// TwinCAT 3 PLC project PLC
// ProgramVersion: 3.1.4026.17
// libraries:
//   Tc2_EtherCAT, * (Beckhoff Automation GmbH)
//   Tc2_Standard, * (Beckhoff Automation GmbH)
//   Tc2_System, * (Beckhoff Automation GmbH)
//   Tc3_Module, * (Beckhoff Automation GmbH)
//   VisuDialogs, * (System)
// project tree:
//   DUTs/00_MainBlocks/ E_SystemStartupSequence.TcDUT
//   DUTs/30_EtherCatDiagnostic/ E_EcDiacStatus.TcDUT (not stored), E_EcGetSlaveName.TcDUT (not stored), E_EcSystemStatus.TcDUT (not stored), ST_EcTerminalDiagInfo.TcDUT (not stored)
//   / GlobalTextList.TcGTLO, ImagePool.TcIPO (not stored), PlcTask.TcTTO, Visualization Manager.TcVMO (not stored), VISU_TASK.TcTTO
//   GVLs/ GVL00_IO.TcGVL, GVL10_VAR_PRG.TcGVL, GVL30_DiagnosticEtherCAT.TcGVL
//   POUs/00_MainBlocks/ MAIN.TcPOU
//   POUs/10_GeneralPlcBlocks/ Blinker.TcPOU, ClockGenerator.TcPOU
//   POUs/10_GeneralPlcBlocks/Components/ FB_Blinker.TcPOU, F_ScaleToByteBeam.TcPOU, F_Scaling.TcPOU
//   POUs/11_TemperatureControl/ TemperatureControl.TcPOU
//   POUs/30_EtherCatDiagnose/Components/ FB_DiagnosticEtherCAT.TcPOU (not stored)
//   POUs/30_EtherCatDiagnose/ DiagnosticEtherCAT.TcPOU (not stored)
//   VISUs/ HmiEtherCatDiagnostic.TcVIS, HmiStartPage.TcVIS
// real-time tasks:
//   TASK PlcTask: cycle T#10ms, priority 20, ADS port 350
//   TASK VISU_TASK: cycle T#200000us, priority 30, ADS port 351
// motion (NC):
//   TASK NC-Task 1 SAF: cycle T#2ms, priority 4, ADS port 501
//   TASK NC-Task 1 SVB: cycle T#10ms, priority 8, ADS port 511
//   AXIS Axis 1 (id 1)
//     OtherSettings: AllowMotionCmdToSlave=true
//     encoder EncType=4
//       EncPara: MaxCount=#x0000ffff
//     drive DrvType=23
//       Analog: TorqueSetpointScale=10, ScaleFactorActTorque=0.1
//       TimeComp: TaskDelayCycles=1
//     controller CtrType=1
//       CtrPara: PriorControlFactor=1
//         Observer: BandWidth=20
//   AXIS Axis 2 (id 2)
//     OtherSettings: AllowMotionCmdToSlave=true
//     encoder EncType=4
//       EncPara: MaxCount=#x0000ffff
//     drive DrvType=23
//       Analog: TorqueSetpointScale=10, ScaleFactorActTorque=0.1
//       TimeComp: TaskDelayCycles=1
//     controller CtrType=1
//       CtrPara: PriorControlFactor=1
//         Observer: BandWidth=20
// I/O:
//   DEVICE Device 2 (EtherCAT), AmsNetId 5.52.100.160.3.1
//     Term 1 (EK1200) [EK1200-5000 EtherCAT Power supply (2A E-Bus)]
//       Term 2 (EL1859) [EL1859 8Ch. Dig. Input 24V, 3ms, 8Ch. Dig. Output 24V, 0.5A]
//       Term 3 (EL1859) [EL1859 8Ch. Dig. Input 24V, 3ms, 8Ch. Dig. Output 24V, 0.5A]
//       Term 4 (EL1004) [EL1004 4Ch. Dig. Input 24V, 3ms]
//       Term 5 (EL2034) [EL2034 4Ch. Dig. Output 24V, 2A, Diagnostic]
//       Term 6 (EL3255) [EL3255 5Ch. potentiometer measurement with sensor supply]
//       Term 7 (EL5151) [EL5151 1Ch. Inc. Encoder]
//       Term 8 (EL3318) [EL3318 8Ch. Ana Input Thermocouple (TC)]
//       Term 9 (EL7332) [EL7332 2Ch. DC motor output stage (24V, 1.5A)]
//       Term 10 (EL3443) [EL3443 3Ch. Power Measuring]
//       Term 11 (EL9011) [EL9011 End Terminal]
// variable links:
//   PLC/PLC Instance <-> Device 2 (EtherCAT)/Term 1 (EK1200)/Term 10 (EL3443)
//     PlcTask Inputs/GVL00_IO.fCurrentFan <-> L3 Basic/Current
//     PlcTask Inputs/GVL00_IO.fCurrentHeating1 <-> L1 Basic/Current
//     PlcTask Inputs/GVL00_IO.fCurrentHeating2 <-> L2 Basic/Current
//     PlcTask Inputs/GVL00_IO.fVoltageFan <-> L3 Basic/Voltage
//     PlcTask Inputs/GVL00_IO.fVoltageHeating1 <-> L1 Basic/Voltage
//     PlcTask Inputs/GVL00_IO.fVoltageHeating2 <-> L2 Basic/Voltage
//   PLC/PLC Instance <-> Device 2 (EtherCAT)/Term 1 (EK1200)/Term 2 (EL1859)
//     PlcTask Inputs/GVL00_IO.bSwitchS10 <-> Channel 1/Input
//     PlcTask Inputs/GVL00_IO.bSwitchS11 <-> Channel 2/Input
//     PlcTask Inputs/GVL00_IO.bSwitchS12 <-> Channel 3/Input
//     PlcTask Inputs/GVL00_IO.bSwitchS13 <-> Channel 4/Input
//     PlcTask Inputs/GVL00_IO.bSwitchS14 <-> Channel 5/Input
//     PlcTask Inputs/GVL00_IO.bSwitchS15 <-> Channel 6/Input
//     PlcTask Inputs/GVL00_IO.bSwitchS16 <-> Channel 7/Input
//     PlcTask Inputs/GVL00_IO.bSwitchS17 <-> Channel 8/Input
//     PlcTask Outputs/GVL00_IO.bLedH10 <-> Channel 9/Output
//     PlcTask Outputs/GVL00_IO.bLedH11 <-> Channel 10/Output
//     PlcTask Outputs/GVL00_IO.bLedH12 <-> Channel 11/Output
//     PlcTask Outputs/GVL00_IO.bLedH13 <-> Channel 12/Output
//     PlcTask Outputs/GVL00_IO.bLedH14 <-> Channel 13/Output
//     PlcTask Outputs/GVL00_IO.bLedH15 <-> Channel 14/Output
//     PlcTask Outputs/GVL00_IO.bLedH16 <-> Channel 15/Output
//     PlcTask Outputs/GVL00_IO.bLedH17 <-> Channel 16/Output
//   PLC/PLC Instance <-> Device 2 (EtherCAT)/Term 1 (EK1200)/Term 3 (EL1859)
//     PlcTask Inputs/GVL00_IO.bSwitchS20 <-> Channel 1/Input
//     PlcTask Inputs/GVL00_IO.bSwitchS21 <-> Channel 2/Input
//     PlcTask Inputs/GVL00_IO.bSwitchS22 <-> Channel 3/Input
//     PlcTask Inputs/GVL00_IO.bSwitchS23 <-> Channel 4/Input
//     PlcTask Inputs/GVL00_IO.bSwitchS24 <-> Channel 5/Input
//     PlcTask Inputs/GVL00_IO.bSwitchS25 <-> Channel 6/Input
//     PlcTask Inputs/GVL00_IO.bSwitchS26 <-> Channel 7/Input
//     PlcTask Inputs/GVL00_IO.bSwitchS27 <-> Channel 8/Input
//     PlcTask Outputs/GVL00_IO.bLedH20 <-> Channel 9/Output
//     PlcTask Outputs/GVL00_IO.bLedH21 <-> Channel 10/Output
//     PlcTask Outputs/GVL00_IO.bLedH22 <-> Channel 11/Output
//     PlcTask Outputs/GVL00_IO.bLedH23 <-> Channel 12/Output
//     PlcTask Outputs/GVL00_IO.bLedH24 <-> Channel 13/Output
//     PlcTask Outputs/GVL00_IO.bLedH25 <-> Channel 14/Output
//     PlcTask Outputs/GVL00_IO.bLedH26 <-> Channel 15/Output
//     PlcTask Outputs/GVL00_IO.bLedH27 <-> Channel 16/Output
//   PLC/PLC Instance <-> Device 2 (EtherCAT)/Term 1 (EK1200)/Term 4 (EL1004)
//     PlcTask Inputs/GVL00_IO.bHeating1Aktiv <-> Channel 1/Input
//     PlcTask Inputs/GVL00_IO.bHeating2Aktiv <-> Channel 2/Input
//   PLC/PLC Instance <-> Device 2 (EtherCAT)/Term 1 (EK1200)/Term 5 (EL2034)
//     PlcTask Outputs/GVL00_IO.bHeating1 <-> Channel 1/Output
//     PlcTask Outputs/GVL00_IO.bHeating2 <-> Channel 2/Output
//     PlcTask Outputs/GVL00_IO.bHeating1Led <-> Channel 3/Output
//     PlcTask Outputs/GVL00_IO.bHeating2Led <-> Channel 4/Output
//   PLC/PLC Instance <-> Device 2 (EtherCAT)/Term 1 (EK1200)/Term 6 (EL3255)
//     PlcTask Inputs/GVL00_IO.nAnalogInR10 <-> AI Standard Channel 1/Value
//     PlcTask Inputs/GVL00_IO.nAnalogInR11 <-> AI Standard Channel 2/Value
//   PLC/PLC Instance <-> Device 2 (EtherCAT)/Term 1 (EK1200)/Term 7 (EL5151)
//     PlcTask Inputs/GVL00_IO.bHandwheelSwitchS18 <-> ENC Inputs/Status/Status of extern latch
//     PlcTask Inputs/GVL00_IO.nHandwheelCounter <-> ENC Inputs/Counter value
//   PLC/PLC Instance <-> Device 2 (EtherCAT)/Term 1 (EK1200)/Term 8 (EL3318)
//     PlcTask Inputs/GVL00_IO.nTemperatureAmbient <-> TC Channel 5/Value
//     PlcTask Inputs/GVL00_IO.nTemperatureCoverHeating <-> TC Channel 4/Value
//     PlcTask Inputs/GVL00_IO.nTemperatureHeatSink <-> TC Channel 3/Value
//     PlcTask Inputs/GVL00_IO.nTemperatureHeating1 <-> TC Channel 1/Value
//     PlcTask Inputs/GVL00_IO.nTemperatureHeating2 <-> TC Channel 2/Value
//   PLC/PLC Instance <-> Device 2 (EtherCAT)/Term 1 (EK1200)/Term 9 (EL7332)
//     PlcTask Inputs/GVL00_IO.nFanStatus <-> DCM Status Channel 1/Status
//     PlcTask Outputs/GVL00_IO.nFanContol <-> DCM Control Channel 1/Control
//     PlcTask Outputs/GVL00_IO.nVeloFan <-> DCM Velocity Channel 1/Velocity

CONFIGURATION PLC
    RESOURCE PLC ON TwinCAT3
        TASK PlcTask(INTERVAL := T#10ms, PRIORITY := 20);
        TASK VISU_TASK(INTERVAL := T#200000us, PRIORITY := 30);
        PROGRAM MAIN WITH PlcTask : MAIN;
        PROGRAM VisuElems_Visu_Prg WITH VISU_TASK : VisuElems.Visu_Prg;
    END_RESOURCE
END_CONFIGURATION

// ---- DUTs/00_MainBlocks/E_SystemStartupSequence.TcDUT
TYPE E_SystemStartupSequence :
(

	eSystemStart_Start						:= 0,
	eSystemStart_Init						:= 10,
	eSystemStart_LedOn						:= 100,
	eSystemStart_LedOff						,
	eSystemStart_Done						:= 500,
	eSystemStart_ErrorStep 					:= 999,
	eSystemStart_NoError
	
);
END_TYPE
(* End *)

// ---- GVLs/GVL00_IO.TcGVL
(* GVL00_IO *)
{attribute 'TcContextName' := 'PlcTask'}
VAR_GLOBAL

	(* EL1859 digital inputs and outputs *)
	{attribute 'OPC.UA.DA' := '1'}
	bSwitchS10						AT%I*	:BOOL;		(* Switch S10 - heating 1 on/off *)
	{attribute 'OPC.UA.DA' := '1'}
	bSwitchS11						AT%I*	:BOOL;		(* Switch S11 - heating 2 on/off *)
	{attribute 'OPC.UA.DA' := '1'}
	bSwitchS12						AT%I*	:BOOL;		(* Switch S12 - fan on/off *)
	{attribute 'OPC.UA.DA' := '1'}
	bSwitchS13						AT%I*	:BOOL;		(* Switch S13 - blinker 1 on/off *)
	{attribute 'OPC.UA.DA' := '1'}
	bSwitchS14						AT%I*	:BOOL;		(* Switch S14 - blinker 2 on/off *)
	{attribute 'OPC.UA.DA' := '1'}
	bSwitchS15						AT%I*	:BOOL;		(* Switch S15 - clock signal 500ms on/off*)
	{attribute 'OPC.UA.DA' := '1'}
	bSwitchS16						AT%I*	:BOOL;		(* Switch S16 - clock signal 1s on/off*)
	{attribute 'OPC.UA.DA' := '1'}
	bSwitchS17						AT%I*	:BOOL;		(* Switch S17 - clock signal 2s on/off*)
	
	{attribute 'OPC.UA.DA' := '1'}
	bLedH10							AT%Q*	:BOOL;		(* LED H10 - heating 1 on *)
	{attribute 'OPC.UA.DA' := '1'}
	bLedH11							AT%Q*	:BOOL;		(* LED H11 - heating 2 on *)
	{attribute 'OPC.UA.DA' := '1'}
	bLedH12							AT%Q*	:BOOL;		(* LED H12 - fan 1 on *)
	{attribute 'OPC.UA.DA' := '1'}
	bLedH13							AT%Q*	:BOOL;		(* LED H13 - blinker 1 *)
	{attribute 'OPC.UA.DA' := '1'}
	bLedH14							AT%Q*	:BOOL;		(* LED H14 - blinker 2 *)
	{attribute 'OPC.UA.DA' := '1'}
	bLedH15							AT%Q*	:BOOL;		(* LED H15 - clock signal 500ms *)
	{attribute 'OPC.UA.DA' := '1'}
	bLedH16							AT%Q*	:BOOL;		(* LED H16 - clock signal 1s *)
	{attribute 'OPC.UA.DA' := '1'}
	bLedH17							AT%Q*	:BOOL;		(* LED H17 - clock signal 2s *)

	(* EL1859 digital inputs/outputs *)
	{attribute 'OPC.UA.DA' := '1'}
	bSwitchS20						AT%I*	:BOOL;		(* Switch S20 - not in use *)
	{attribute 'OPC.UA.DA' := '1'}
	bSwitchS21						AT%I*	:BOOL;		(* Switch S21 - not in use *)
	{attribute 'OPC.UA.DA' := '1'}
	bSwitchS22						AT%I*	:BOOL;		(* Switch S22 - not in use *)
	{attribute 'OPC.UA.DA' := '1'}
	bSwitchS23						AT%I*	:BOOL;		(* Switch S23 - not in use *)
	{attribute 'OPC.UA.DA' := '1'}
	bSwitchS24						AT%I*	:BOOL;		(* Switch S24 - not in use *)
	{attribute 'OPC.UA.DA' := '1'}
	bSwitchS25						AT%I*	:BOOL;		(* Switch S25 - not in use *)
	{attribute 'OPC.UA.DA' := '1'}
	bSwitchS26						AT%I*	:BOOL;		(* Switch S26 - not in use *)
	{attribute 'OPC.UA.DA' := '1'}
	bSwitchS27						AT%I*	:BOOL;		(* Switch S27 - not in use *)

	{attribute 'OPC.UA.DA' := '1'}
	bLedH20							AT%Q*	:BOOL;		(* LED H20 - temperature heat sink >23.75C° *)
	{attribute 'OPC.UA.DA' := '1'}
	bLedH21							AT%Q*	:BOOL;		(* LED H21 - temperature heat sink >27.50C° *)
	{attribute 'OPC.UA.DA' := '1'}
	bLedH22							AT%Q*	:BOOL;		(* LED H22 - temperature heat sink >31,25C° *)
	{attribute 'OPC.UA.DA' := '1'}
	bLedH23							AT%Q*	:BOOL;		(* LED H23 - temperature heat sink >35.00C° *)
	{attribute 'OPC.UA.DA' := '1'}
	bLedH24							AT%Q*	:BOOL;		(* LED H24 - temperature heat sink >38.75C° *)
	{attribute 'OPC.UA.DA' := '1'}
	bLedH25							AT%Q*	:BOOL;		(* LED H25 - temperature heat sink >42.50C° *)
	{attribute 'OPC.UA.DA' := '1'}
	bLedH26							AT%Q*	:BOOL;		(* LED H26 - temperature heat sink >46.25C° *)
	{attribute 'OPC.UA.DA' := '1'}
	bLedH27							AT%Q*	:BOOL;		(* LED H27 - temperature heat sink >50.00C° *)

	(* EL1004 digital inputs *)
	{attribute 'OPC.UA.DA' := '1'}
	bHeating1Aktiv					AT%I*	:BOOL;		(* Heating 1 aktiv *)
	{attribute 'OPC.UA.DA' := '1'}
	bHeating2Aktiv					AT%I*	:BOOL;		(* Heating 2 aktiv *)

	(* EL2034 digital outputs *)
	{attribute 'OPC.UA.DA' := '1'}
	bHeating1						AT%Q*	:BOOL;		(* Heating 1 *)
	{attribute 'OPC.UA.DA' := '1'}
	bHeating2						AT%Q*	:BOOL;		(* Heating 2 *)
	{attribute 'OPC.UA.DA' := '1'}
	bHeating1Led					AT%Q*	:BOOL;		(* Heating 1 Led - flash slow (temperature > 40.0) - flash fast (temperature > 45.0) *)
	{attribute 'OPC.UA.DA' := '1'}
	bHeating2Led					AT%Q*	:BOOL;		(* Heating 2 Led - flash slow (temperature > 40.0) - flash fast (temperature > 45.0) *)

	(* EL3255 0..10V analog inputs *)
	{attribute 'OPC.UA.DA' := '1'}
	nAnalogInR10					AT%I*	:INT;		(* Analog input R10 - fan velocity *)
	{attribute 'OPC.UA.DA' := '1'}
	nAnalogInR11					AT%I*	:INT;		(* Analog input R11 - blinker 1 flash speed *)
	
	(* EL5151 incremental encoder 24 increments/rotation * 4-fold evaluation -> 96  increments/rotation*)
	{attribute 'OPC.UA.DA' := '1'}
	nHandwheelCounter				AT%I*	:UINT;		(* handwheel counter *)
	{attribute 'OPC.UA.DA' := '1'}
	bHandwheelSwitchS18				AT%I*	:BOOL;		(* Switch S18 *)	
	
	(* EL3318 8-channel thermocouple inputs *)
	{attribute 'OPC.UA.DA' := '1'}
	nTemperatureHeating1			AT%I*	:INT;		(* Temperature heating 1 *)
	{attribute 'OPC.UA.DA' := '1'}
	nTemperatureHeating2			AT%I*	:INT;		(* Temperature heating 2 *)
	{attribute 'OPC.UA.DA' := '1'}
	nTemperatureHeatSink			AT%I*	:INT;		(* Temperature heat sink *)
	{attribute 'OPC.UA.DA' := '1'}
	nTemperatureCoverHeating		AT%I*	:INT;		(* Temperature cover heating *)
	{attribute 'OPC.UA.DA' := '1'}
	nTemperatureAmbient				AT%I*	:INT;		(* Temperature ambient *)
	
	(* EL7332 2-channel DC motor output stage - fan *)
	{attribute 'OPC.UA.DA' := '1'}
	nFanStatus						AT%I*	:UINT;		(* Fan status *)
	{attribute 'OPC.UA.DA' := '1'}
	nVeloFan						AT%Q*	:INT;		(* Fan velocity*)
	{attribute 'OPC.UA.DA' := '1'}
	nFanContol						AT%Q*	:UINT;		(* Fan control *)

	(* EL3443 3-phase power measurement terminal *)
	{attribute 'OPC.UA.DA' := '1'}
	fVoltageHeating1				AT%I*	:REAL;		(* Voltage heating 1 (V)*)
	{attribute 'OPC.UA.DA' := '1'}
	fCurrentHeating1				AT%I*	:REAL;		(* Current heating 1 (A)*)
	{attribute 'OPC.UA.DA' := '1'}
	fVoltageHeating2				AT%I*	:REAL;		(* Voltage heating 1 (V)*)
	{attribute 'OPC.UA.DA' := '1'}
	fCurrentHeating2				AT%I*	:REAL;		(* Current heating 1 (A)*)
	{attribute 'OPC.UA.DA' := '1'}
	fVoltageFan						AT%I*	:REAL;		(* Voltage fan 1 (V)*)
	{attribute 'OPC.UA.DA' := '1'}
	fCurrentFan						AT%I*	:REAL;		(* Current fan 1 (power converter 1:32) (A*32) *)
	
END_VAR
(* End *)

// ---- GVLs/GVL10_VAR_PRG.TcGVL
(* Variables for program blocks *)
VAR_GLOBAL

	(* PLC start detected *)
	bFirstCycleDetected						:BOOL;
	bMachineSequenzAktiv					:BOOL;		(* PLC startup done (LED test) program in cyclic mode *)

	(* Clock generator *)
	bClock500ms								:BOOL;		(* Clock 500ms on/off *)
	bClock1s								:BOOL;		(* Clock 1s on/off *)
	bClock2s								:BOOL;		(* Clock 2s on/off *)
	bRisingEdge500ms						:BOOL;		(* Rising edge all 500ms over one cycle *)
	bRisingEdge1s							:BOOL;		(* Edge after 1s over a cycle *)
	bRisingEdge2s							:BOOL;		(* Edge after 2s over a cycle *)

END_VAR
(* End *)

// ---- GVLs/GVL30_DiagnosticEtherCAT.TcGVL
(* GVL30_DiagnosticEtherCAT *)
{attribute 'TcContextName' := 'PlcTask'}
VAR_GLOBAL

	fbDiagnosticEtherCAT					:FB_DiagnosticEtherCAT;

END_VAR
(* End *)

// ---- POUs/00_MainBlocks/MAIN.TcPOU
PROGRAM MAIN
(*******************************************************************************************************
Title				:	Main program 
Description			:	Calling the created subroutines (Task 1ms)
Version / Date		:	1.0.0 / 12.02.2018 / created program (Version progress see below)

Supported hardware	: 	Demo-Rack mobile IoT

Used Documentation	:	
Documentation	
Version/Date 		:	

Required libraries 	: 	Please look in the "References" folder
********************************************************************************************************)
VAR
	
(* Cycle counter *)
	nCycleCounter							:UDINT;

(* act_SystemStart *)
	eStateSystemStartSeq					:E_SystemStartupSequence;
	eSystemStartSeqErrStep					:E_SystemStartupSequence := eSystemStart_NoError;
	bSystemStartErr							:BOOL;
	bSystemStartEnd							:BOOL;
	fbTimerSystemStart						:TON;

END_VAR
(*******************************************************************************************************
Version / Date / Description:
1.0.0   / 12.02.2018 / created program
********************************************************************************************************)
(* End *)

(* MAIN - 1ms *)

(* THIS CODE IS ONLY AN EXAMPLE - YOU HAVE TO CHECK APTITUDE FOR YOUR APPLICATION *)

(* Cycle counter *)
	nCycleCounter := nCycleCounter + 1;


(* Startup detect *)
	IF TwinCAT_SystemInfoVarList._TaskInfo[GETCURTASKINDEXEX()].FirstCycle
	THEN
		bFirstCycleDetected	:= TRUE;
	END_IF


(* Startup- or machine sequence *)
	IF bFirstCycleDetected
	THEN
	(* Startup sequenz *)
		act_SystemStart();

		IF bSystemStartEnd
		THEN
			bFirstCycleDetected := FALSE;
			bMachineSequenzAktiv := TRUE;
		END_IF

	ELSIF bMachineSequenzAktiv
	THEN
	(* Machine sequenz *)

		(* Test clock generator *)
			ClockGenerator();	
			
		(* Test blinker *)
			Blinker();
			
		(* Test temperature control *)
			TemperatureControl();

		(* Test EtherCAT diacnostic *)
			DiagnosticEtherCAT();

	END_IF

(* End *)

ACTION act_SystemStart:
(* Aktion system start *)

	CASE eStateSystemStartSeq OF

	
		eSystemStart_Start			: 	(* Waiting for start *)
		
				eStateSystemStartSeq := eSystemStart_Init;

				
		eSystemStart_Init			:	(* Initialize *)

				fbTimerSystemStart(IN := FALSE);
				eStateSystemStartSeq := eSystemStart_LedOn;

				
		eSystemStart_LedOn			:	(* Sequence Leds on *)

				fbTimerSystemStart(	
					IN := TRUE,
					PT := T#2250MS);

				bLedH10	:=	fbTimerSystemStart.ET > T#250MS;
				bLedH20 :=  bLedH10;
				bLedH11	:=	fbTimerSystemStart.ET > T#500MS;
				bLedH21 :=  bLedH11;
				bLedH12	:=	fbTimerSystemStart.ET > T#750MS;
				bLedH22 :=  bLedH12;
				bLedH13	:=	fbTimerSystemStart.ET > T#1000MS;
				bLedH23 :=  bLedH13;
				bLedH14	:=	fbTimerSystemStart.ET > T#1250MS;
				bLedH24 :=  bLedH14;
				bLedH15	:=	fbTimerSystemStart.ET > T#1500MS;
				bLedH25 :=  bLedH15;
				bLedH16	:=	fbTimerSystemStart.ET > T#1750MS;
				bLedH26 :=  bLedH16;
				bLedH17	:=	fbTimerSystemStart.ET > T#2000MS;
				bLedH27 :=  bLedH17;

				IF fbTimerSystemStart.Q
				THEN
					fbTimerSystemStart(IN := FALSE);
					eStateSystemStartSeq := eSystemStart_LedOff;
				ELSIF FALSE
				THEN
					(* If error then notice the step *)
					eSystemStartSeqErrStep := eStateSystemStartSeq;
					eStateSystemStartSeq   := eSystemStart_ErrorStep;
				END_IF

				
		eSystemStart_LedOff			:	(* Sequence Leds off *)

				fbTimerSystemStart(	
					IN := TRUE,
					PT := T#2250MS);

				bLedH10	:=	fbTimerSystemStart.ET < T#250MS;
				bLedH20 :=  bLedH10;
				bLedH11	:=	fbTimerSystemStart.ET < T#500MS;
				bLedH21 :=  bLedH11;
				bLedH12	:=	fbTimerSystemStart.ET < T#750MS;
				bLedH22 :=  bLedH12;
				bLedH13	:=	fbTimerSystemStart.ET < T#1000MS;
				bLedH23 :=  bLedH13;
				bLedH14	:=	fbTimerSystemStart.ET < T#1250MS;
				bLedH24 :=  bLedH14;
				bLedH15	:=	fbTimerSystemStart.ET < T#1500MS;
				bLedH25 :=  bLedH15;
				bLedH16	:=	fbTimerSystemStart.ET < T#1750MS;
				bLedH26 :=  bLedH16;
				bLedH17	:=	fbTimerSystemStart.ET < T#2000MS;
				bLedH27 :=  bLedH17;
									
				IF fbTimerSystemStart.Q
				THEN
					eStateSystemStartSeq := eSystemStart_Done;
				ELSIF FALSE
				THEN
					(* If error then notice the step *)
					eSystemStartSeqErrStep := eStateSystemStartSeq;
					eStateSystemStartSeq   := eSystemStart_ErrorStep;
				END_IF

				
		eSystemStart_Done			:	(* System start done *)

				bSystemStartEnd := TRUE;

				
		eSystemStart_ErrorStep		:	(* Error on system start *)

				bSystemStartErr := TRUE;

				IF FALSE
				THEN
					bSystemStartErr        := FALSE;
					eSystemStartSeqErrStep := eSystemStart_NoError;
					eStateSystemStartSeq   := eSystemStart_Start;
				END_IF 

	ELSE
		
		(* If not a valid step is active, then put on start *)
		eSystemStartSeqErrStep := eSystemStart_NoError;
		eStateSystemStartSeq   := eSystemStart_Start;
	
	END_CASE

(* End *)
END_ACTION

END_PROGRAM

// ---- POUs/10_GeneralPlcBlocks/ClockGenerator.TcPOU
PROGRAM ClockGenerator
VAR
	
	nCycleTime								:UDINT;		(* Cycle time from the PLC Task *)
	nTimeValue								:INT;		(* Time value clock generator*)
	
END_VAR
(* End *)

(* Clock generator *)

	(* PLC cycle time in ms  *)
	nCycleTime	:=	TwinCAT_SystemInfoVarList._TaskInfo[GETCURTASKINDEXEX()].cycleTime / 10000;

	
	(* Calculate with the cycle time the time value *)
	nTimeValue	:=	nTimeValue + UDINT_TO_INT(nCycleTime);

	
	(* Generate the clocks and the rising edges with the time value *)
	CASE nTimeValue OF

		500		:	bClock500ms			:=	TRUE;
					bRisingEdge500ms	:=	TRUE;

		1000	:	bClock500ms			:=	FALSE;
					bRisingEdge500ms	:=	TRUE;
					bClock1s			:=	TRUE;
					bRisingEdge1s		:=	TRUE;

		1500	:	bClock500ms			:=	TRUE;
					bRisingEdge500ms	:=	TRUE;

		2000	:	bClock500ms			:=	FALSE;
					bRisingEdge500ms	:=	TRUE;
					bClock1s			:=	FALSE;
					bRisingEdge1s		:=	TRUE;
					bClock2s			:=	TRUE;
					bRisingEdge2s		:=	TRUE;

		2500	:	bClock500ms			:=	TRUE;
					bRisingEdge500ms	:=	TRUE;

		3000	:	bClock500ms			:=	FALSE;
					bRisingEdge500ms	:=	TRUE;
					bClock1s			:=	TRUE;
					bRisingEdge1s		:=	TRUE;

		3500	:	bClock500ms			:=	TRUE;
					bRisingEdge500ms	:=	TRUE;

		4000	:	bClock500ms			:=	FALSE;
					bRisingEdge500ms	:=	TRUE;
			 		bClock1s			:=	FALSE;
					bRisingEdge1s		:=	TRUE;
					bClock2s			:=	FALSE;
					bRisingEdge2s		:=	TRUE;
					
	ELSE

		(* Reset the rising edge variables after one cycle *)
		bRisingEdge500ms	:=	FALSE;
		bRisingEdge1s		:=	FALSE;
		bRisingEdge2s		:=	FALSE;

	END_CASE;

	
	(* Sequence reset at 4000ms *)
	IF nTimeValue >= 4000
	THEN
		nTimeValue := 0;
	END_IF
	

	(* Outputs *)
	bLedH15 := bSwitchS15 AND bClock500ms;
	bLedH16 := bSwitchS16 AND bClock1s;
	bLedH17 := bSwitchS17 AND bClock2s;


(* End *)

END_PROGRAM

// ---- POUs/10_GeneralPlcBlocks/Blinker.TcPOU
PROGRAM Blinker
VAR
	
	fbBlinker1								:FB_Blinker;
	tTurnOffDelayB1							:TIME := T#1S;
	fbBlinker2								:FB_Blinker;
	
END_VAR
(* End *)

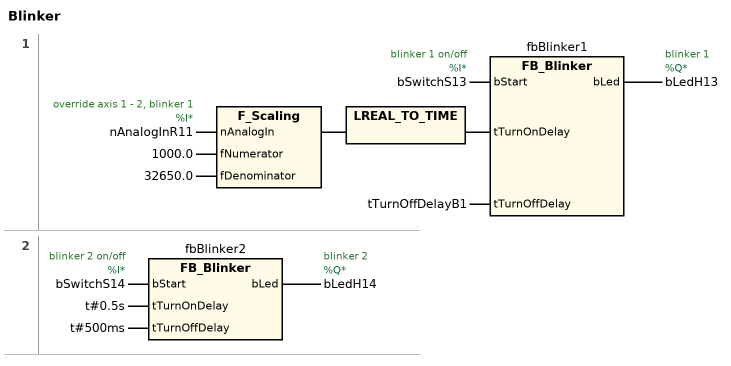
// NETWORK 1
//   bSwitchS13: blinker 1 on/off | AT %I*
//   nAnalogInR11: override axis 1 - 2, blinker 1 | AT %I*
//   bLedH13: blinker 1 | AT %Q*
fbBlinker1(
    bStart := bSwitchS13,
    tTurnOnDelay := LREAL_TO_TIME(F_Scaling(nAnalogIn := nAnalogInR11, fNumerator := 1000.0, fDenominator := 32650.0)),
    tTurnOffDelay := tTurnOffDelayB1); // FB_Blinker
bLedH13 := fbBlinker1.bLed;

// NETWORK 2
//   bSwitchS14: blinker 2 on/off | AT %I*
//   bLedH14: blinker 2 | AT %Q*
fbBlinker2(bStart := bSwitchS14, tTurnOnDelay := t#0.5s, tTurnOffDelay := t#500ms); // FB_Blinker
bLedH14 := fbBlinker2.bLed;

END_PROGRAM

// ---- POUs/10_GeneralPlcBlocks/Components/FB_Blinker.TcPOU
FUNCTION_BLOCK FB_Blinker
VAR_INPUT

	bStart									:BOOL;
	tTurnOnDelay							:TIME;
	tTurnOffDelay							:TIME;

END_VAR
VAR_OUTPUT

	bLed									:BOOL;

END_VAR
VAR

	fbTimer1								:TON;
	fbTimer2								:TON;

END_VAR
(* End *)

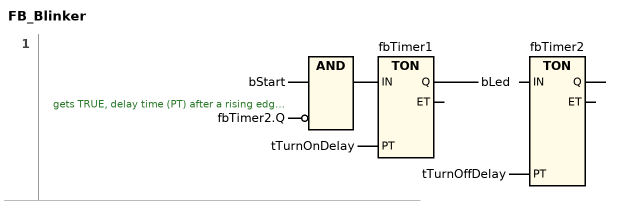
// NETWORK 1
//   fbTimer2.Q: gets TRUE, delay time (PT) after a rising edge at IN
fbTimer1(IN := bStart AND NOT fbTimer2.Q, PT := tTurnOnDelay); // TON
bLed := fbTimer1.Q;
fbTimer2(IN := fbTimer1.Q, PT := tTurnOffDelay); // TON

END_FUNCTION_BLOCK

// ---- POUs/10_GeneralPlcBlocks/Components/F_Scaling.TcPOU
FUNCTION F_Scaling : LREAL
VAR_INPUT

	nAnalogIn								:INT;
	fNumerator								:LREAL;
	fDenominator							:LREAL;
	
END_VAR
VAR
END_VAR
(* End *)

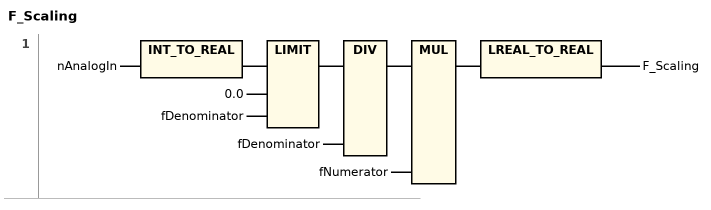
// NETWORK 1
F_Scaling := LREAL_TO_REAL((LIMIT(INT_TO_REAL(nAnalogIn), 0.0, fDenominator) / fDenominator) * fNumerator);

END_FUNCTION

// ---- POUs/11_TemperatureControl/TemperatureControl.TcPOU
PROGRAM TemperatureControl
VAR

	(* Temperatures *)
	fTemperatureCHeating1					:REAL;		(* Temperature heating 1 (C°)*)
	fTemperatureCHeating2					:REAL;		(* Temperature heating 2 (C°)*)
	fTemperatureCHeatSink					:REAL;		(* Temperature heat sink (C°)*)
	nTemperatureHeatSinkLedArray			:BYTE;		(* Temperature heat sink - 8 Led array *)
	fTemperatureCCoverHeating				:REAL;		(* Temperature cover heating (C°)*)
	fTemperatureCAmbient					:REAL;		(* Temperature ambient (C°)*)

	(* Fan *)
	fCurrentFanA							:REAL;		(* Current fan 1 (A)*)	
	fVeloFanProcent							:LREAL;		(* Fan velocity (%)*)
	
END_VAR
(* End *)

(* Temperature control *)
 

(* Scaling temperature variables *)
	fTemperatureCHeating1 	     := TO_REAL(nTemperatureHeating1) / 10.0;			
	fTemperatureCHeating2 	     := TO_REAL(nTemperatureHeating2) / 10.0;

	fTemperatureCHeatSink 	  	 := TO_REAL(nTemperatureHeatSink) / 10.0;
	nTemperatureHeatSinkLedArray :=	F_ScaleToByteBeam(fActValue:= fTemperatureCHeatSink - 20.0 , fMaxValue:= 30.0);
	bLedH20 := nTemperatureHeatSinkLedArray.0;	(* >23.75C° -> Led on *) 
	bLedH21 := nTemperatureHeatSinkLedArray.1;	(* >27.50C° -> Led on *)
	bLedH22 := nTemperatureHeatSinkLedArray.2;	(* >31,25C° -> Led on *)
	bLedH23 := nTemperatureHeatSinkLedArray.3;	(* >35.00C° -> Led on *)
	bLedH24 := nTemperatureHeatSinkLedArray.4;	(* >38.75C° -> Led on *)
	bLedH25 := nTemperatureHeatSinkLedArray.5;	(* >42.50C° -> Led on *)
	bLedH26 := nTemperatureHeatSinkLedArray.6;	(* >46.25C° -> Led on *)
	bLedH27 := nTemperatureHeatSinkLedArray.7;	(* >50.00C° -> Led on *)

	fTemperatureCCoverHeating    := TO_REAL(nTemperatureCoverHeating) / 10.0;

	fTemperatureCAmbient 	     := TO_REAL(nTemperatureAmbient) / 10.0;

	
(* Heating 1 *)
	bHeating1 := bSwitchS10 
					AND NOT (fTemperatureCHeating1 > 48.0)					(* >48.0C° -> switch off *)
						AND NOT fbDiagnosticEtherCAT.nFrmXWcState[0].1		(* 1 -> Terminals not in communication -> switch off *)
							AND NOT fbDiagnosticEtherCAT.nFrmXWcState[0].2;

	bLedH10 	 := bHeating1Aktiv;
	
	IF (fTemperatureCHeating1 > 45.0) 
	THEN
		bHeating1Led := bClock500ms;
	ELSIF (fTemperatureCHeating1 > 40.0) 
	THEN
		bHeating1Led := bClock2s;
	ELSIF bHeating1Aktiv 
	THEN
		bHeating1Led := TRUE;
	ELSE
		bHeating1Led := FALSE;
	END_IF

	
(* Heating 2 *)
	bHeating2 := bSwitchS11 
					AND NOT (fTemperatureCHeating2 > 48.0)					(* >48.0C° -> switch off *)
						AND NOT fbDiagnosticEtherCAT.nFrmXWcState[0].1		(* 1 -> Terminals not in communication -> switch off *)
							AND NOT fbDiagnosticEtherCAT.nFrmXWcState[0].2;

	bLedH11 := bHeating2Aktiv;
	
	IF (fTemperatureCHeating2 > 45.0) 
	THEN
		bHeating2Led := bClock500ms;
	ELSIF (fTemperatureCHeating2 > 40.0) 
	THEN
		bHeating2Led := bClock2s;
	ELSIF bHeating2Aktiv 
	THEN
		bHeating2Led := TRUE;
	ELSE
		bHeating2Led := FALSE;
	END_IF


(* Fan control *)
	(* Enable fan *)
	nFanContol.0 := bSwitchS12;

	(* Fan ready *)
	bLedH12 	 := nFanStatus.1;

	(* Fan velocity *)	
	nVeloFan 		:= TO_INT(F_Scaling(nAnalogInR10, 19000.0, 32650.0)) + 1000;
	fVeloFanProcent := F_Scaling(nAnalogInR10, 90.0, 32650.0) + 10.0;

	(* Fan actual current (A)*)
	fCurrentFanA	:= fCurrentFan * 32.0;
	
	
(* End *)

END_PROGRAM

// ---- POUs/10_GeneralPlcBlocks/Components/F_ScaleToByteBeam.TcPOU
FUNCTION F_ScaleToByteBeam : Byte
VAR_INPUT
	
	fActValue								:LREAL;
	fMaxValue								:LREAL;
	
END_VAR
VAR
	
	nValueBeam								:BYTE;
	
END_VAR
(* End *)

(* Scale to byte beam *)

	nValueBeam := TO_BYTE(TRUNC(F_Scaling(nAnalogIn:=TO_INT(ABS(fActValue)), fNumerator:=8.0, fDenominator:=fMaxValue )));
	
	CASE nValueBeam OF
		0	:	F_ScaleToByteBeam := 2#0;
		1	:	F_ScaleToByteBeam := 2#1;
		2	:	F_ScaleToByteBeam := 2#11;
		3	:	F_ScaleToByteBeam := 2#111;
		4	:	F_ScaleToByteBeam := 2#1111;
		5	:	F_ScaleToByteBeam := 2#11111;
		6	:	F_ScaleToByteBeam := 2#111111;
		7	:	F_ScaleToByteBeam := 2#1111111;
		8	:	F_ScaleToByteBeam := 2#11111111;
	END_CASE
	
(* End *)

END_FUNCTION

// ---- GlobalTextList.TcGTLO
TEXTLIST GlobalTextList
  71 = '%.1f C'
  353 = '%d'
  356 = '%d   '
  69 = '(S10) %.1f C'
  70 = '(S11) %.1f C'
  72 = '(S12) %.1f pct (R10)'
  249 = 'Addr'
  352 = 'Analog / Handwheel'
  796 = 'EtherCAT\nDIAGNOSTIC'
  68 = 'Handwheel S18:'
  354 = 'Increments'
  251 = 'Name'
  709 = 'Potentiometer R10:'
  355 = 'Potentiometer R11:'
  156 = 'S10'
  157 = 'S11'
  158 = 'S12'
  159 = 'S13'
  160 = 'S14'
  514 = 'S15'
  515 = 'S16'
  516 = 'S17'
  517 = 'S20'
  518 = 'S21'
  519 = 'S22'
  520 = 'S23'
  521 = 'S24'
  522 = 'S25'
  350 = 'S26'
  351 = 'S27'
  304 = 'START PAGE'
  252 = 'Status'
  155 = 'Switches'
  250 = 'Type'
END_TEXTLIST

// ---- VISUs/HmiEtherCatDiagnostic.TcVIS
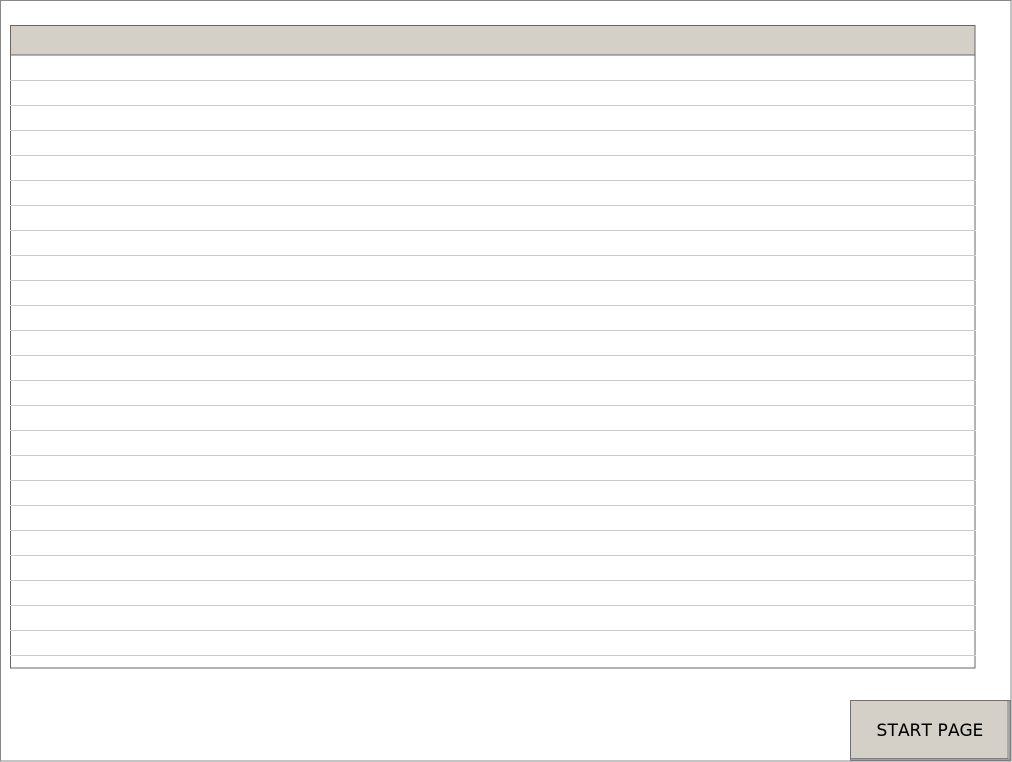
VISUALIZATION HmiEtherCatDiagnostic  // 1012x762
    Button (850,700 160x60), "START PAGE"
        OnMouseClick: change screen: HmiStartPage
    Table (10,25 965x643), data array: fbDiagnosticEtherCAT.stEcTerminalDiagInfo
        p3854506369: fbDiagnosticEtherCAT.stEcTerminalDiagInfo[INDEX].nAddr
        p1892666644: fbDiagnosticEtherCAT.stEcTerminalDiagInfo[INDEX].sType
        p338671338: fbDiagnosticEtherCAT.stEcTerminalDiagInfo[INDEX].sName
        p2170511999: fbDiagnosticEtherCAT.stEcTerminalDiagInfo[INDEX].sTerminalStatus
END_VISUALIZATION

// ---- VISUs/HmiStartPage.TcVIS
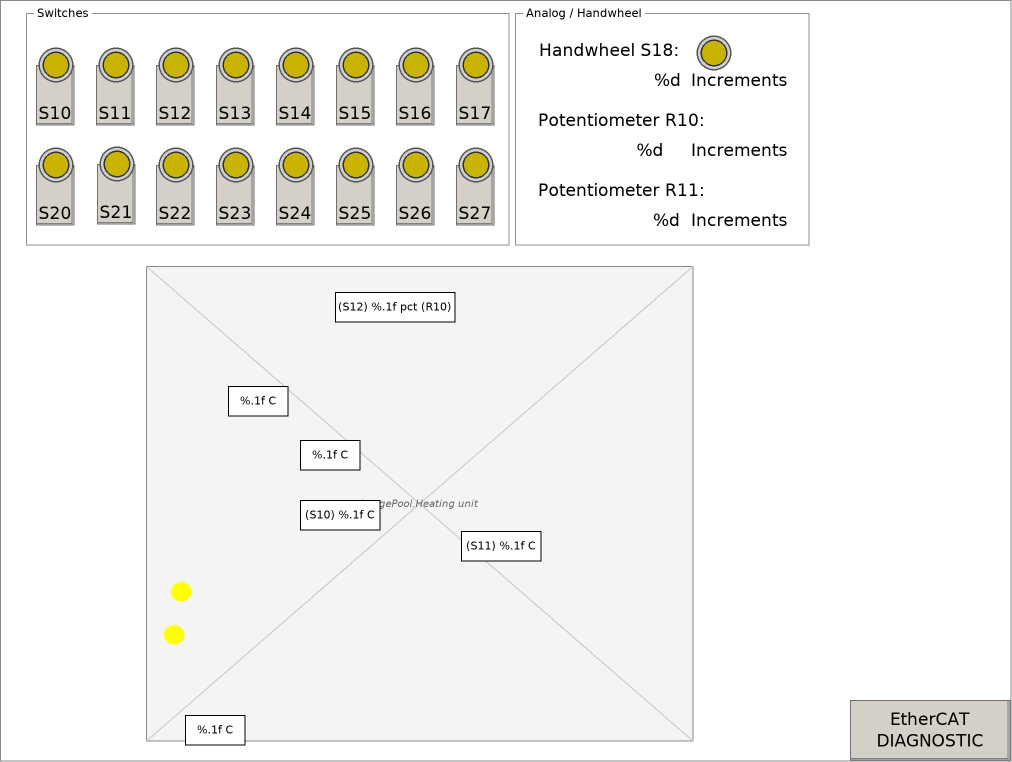
VISUALIZATION HmiStartPage  // 1012x762
    Image (146,266 547x475), image: ImagePool.Heating unit
    Button (850,700 160x60), "EtherCAT DIAGNOSTIC"
        OnMouseClick: change screen: HmiEtherCatDiagnostic
    GroupBox (26,5 483x240), "Switches"
        Button (10,60 38x60), "S10", colour toggle: bSwitchS10
            toggle bSwitchS10
        Lamp1 (10,40 40x40), variable: bLedH10, style: Lamp-Lamp1-Yellow
        Button (70,60 38x60), "S11", colour toggle: bSwitchS11
            toggle bSwitchS11
        Lamp1 (70,40 40x40), variable: bLedH11, style: Lamp-Lamp1-Yellow
        Button (130,60 38x60), "S12", colour toggle: bSwitchS12
            toggle bSwitchS12
        Lamp1 (130,40 40x40), variable: bLedH12, style: Lamp-Lamp1-Yellow
        Button (190,60 38x60), "S13", colour toggle: bSwitchS13
            toggle bSwitchS13
        Lamp1 (190,40 40x40), variable: bLedH13, style: Lamp-Lamp1-Yellow
        Button (250,60 38x60), "S14", colour toggle: bSwitchS14
            toggle bSwitchS14
        Lamp1 (250,40 40x40), variable: bLedH14, style: Lamp-Lamp1-Yellow
        Button (310,60 38x60), "S15", colour toggle: bSwitchS15
            toggle bSwitchS15
        Lamp1 (310,40 40x40), variable: bLedH15, style: Lamp-Lamp1-Yellow
        Button (370,60 38x60), "S16", colour toggle: bSwitchS16
            toggle bSwitchS16
        Lamp1 (370,40 40x40), variable: bLedH16, style: Lamp-Lamp1-Yellow
        Button (430,60 38x60), "S17", colour toggle: bSwitchS17
            toggle bSwitchS17
        Lamp1 (430,40 40x40), variable: bLedH17, style: Lamp-Lamp1-Yellow
        Button (10,160 38x60), "S20", colour toggle: bSwitchS20
            toggle bSwitchS20
        Lamp1 (10,140 40x40), variable: bLedH20, style: Lamp-Lamp1-Yellow
        Button (71,159 38x60), "S21", colour toggle: bSwitchS21
            toggle bSwitchS21
        Lamp1 (71,139 40x40), variable: bLedH21, style: Lamp-Lamp1-Yellow
        Button (130,160 38x60), "S22", colour toggle: bSwitchS22
            toggle bSwitchS22
        Lamp1 (130,140 40x40), variable: bLedH22, style: Lamp-Lamp1-Yellow
        Button (190,160 38x60), "S23", colour toggle: bSwitchS23
            toggle bSwitchS23
        Lamp1 (190,140 40x40), variable: bLedH23, style: Lamp-Lamp1-Yellow
        Button (250,160 38x60), "S24", colour toggle: bSwitchS24
            toggle bSwitchS24
        Lamp1 (250,140 40x40), variable: bLedH24, style: Lamp-Lamp1-Yellow
        Button (310,160 38x60), "S25", colour toggle: bSwitchS25
            toggle bSwitchS25
        Lamp1 (310,140 40x40), variable: bLedH25, style: Lamp-Lamp1-Yellow
        Button (370,160 38x60), "S26", colour toggle: bSwitchS26
            toggle bSwitchS26
        Lamp1 (370,140 40x40), variable: bLedH26, style: Lamp-Lamp1-Yellow
        Button (430,160 38x60), "S27", colour toggle: bSwitchS27
            toggle bSwitchS27
        Lamp1 (430,140 40x40), variable: bLedH27, style: Lamp-Lamp1-Yellow
    GroupBox (515,5 294x240), "Analog / Handwheel"
        Rectangle (20,200 148x30), "%d", text variable: nAnalogInR11
            OnMouseClick: write the text variable via Default, min 0, max 32767
        Label (173,200 118x30), "Increments"
        Label (20,170 197x30), "Potentiometer R11:"
        Rectangle (20,130 148x30), "%d", text variable: nAnalogInR10
            OnMouseClick: write the text variable via Default, min 0, max 32767
        Label (173,130 121x30), "Increments"
        Label (20,100 216x30), "Potentiometer R10:"
        Lamp1 (179,28 40x40), variable: bHandwheelSwitchS18, style: Lamp-Lamp1-Yellow
        Rectangle (21,60 148x30), "%d", text variable: nHandwheelCounter
            OnMouseClick: write the text variable via Default
        Label (173,60 133x30), "Increments"
        Label (21,30 216x30), "Handwheel S18:"
    Rectangle (300,500 80x30), "(S10) %.1f C", text variable: TemperatureControl.fTemperatureCHeating1, colour toggle: bHeating1Aktiv
    Rectangle (461,531 80x30), "(S11) %.1f C", text variable: TemperatureControl.fTemperatureCHeating2, colour toggle: bHeating2Aktiv
    Rectangle (300,440 60x30), "%.1f C", text variable: TemperatureControl.fTemperatureCHeatSink
    Rectangle (228,386 60x30), "%.1f C", text variable: TemperatureControl.fTemperatureCCoverHeating
    Rectangle (185,715 60x30), "%.1f C", text variable: TemperatureControl.fTemperatureCAmbient
    Rectangle (335,292 120x30), "(S12) %.1f pct (R10)", text variable: TemperatureControl.fVeloFanProcent, colour toggle: nFanStatus.1
    Ellipse (171,582 20x19), invisible if: NOT bHeating1Led
    Ellipse (164,625 20x19), invisible if: NOT bHeating2Led
END_VISUALIZATION
